INTERFACE I_MotionInterlocksCommon  EXTENDS I_Error

METHOD DriveCommands
VAR_INPUT
    MoveEnable: BOOL;
    NewMoveReq : BOOL;
END_VAR
END_METHOD

METHOD EnableInterlocks
VAR_INPUT
	UserEnable : BOOL;
	HardwareEnable : BOOL;
END_VAR
END_METHOD

PROPERTY MoveOk : BOOL
GET
END_GET
END_PROPERTY

PROPERTY PowerEnabled : BOOL
GET
END_GET
END_PROPERTY

METHOD Reset
VAR_INPUT
END_VAR
END_METHOD

END_INTERFACE

(* stored: Version 1.1.0.1
   Itf I_MotionInterlocksCommon: Id {6906b881-f15f-4df2-99d8-615248381a43}
   Method DriveCommands: Id {95d7873b-b1cc-491b-828c-b846b0af66ce}
   Method EnableInterlocks: Id {44152237-0773-4dbc-8200-7c97addc3446}
   Property MoveOk: Id {1afd93f7-f2a6-41c4-917d-1b6c9a77ea87}
   Get Get: Id {eb795768-982c-4440-9ee6-002d67c772ee}
   Property PowerEnabled: Id {c51eea5c-413d-4ba5-abaf-3b70155b6bdc}
   Get Get: Id {05bad098-7800-4d94-a94a-923a51852e71}
   Method Reset: Id {cc36a04e-8ae1-4d1a-b6d2-3ef1ada15b9d} *)
